PROGRAM P20_ExhaustFan_old
VAR
		(*****************Wentylator wyciągaowy*******************)
	fbExhaustFan							: FB_MitsubishiInverter;
	fbSensorAcetone							: FB_SensorAcetone;
	fbSensorAirFlow							: FB_SensorFlow;
	
	eExhaustFanState						: E_Station;			
	eExhaustFanRunningState					: E_ConveyorState;	
	fbExhaustFanState						: FB_State;		
	QnExhaustFanVelocitySV					AT %Q*: UDINT; 			(*po kom*)	// Nastawa prędkości transportera
	InExhaustFanVelocityCV 					AT %I*: UDINT;			(*po kom*)
	InExhaustFanSTW 						AT %I*: UINT; 			(*po kom*)	// Statusword transportera wejściowego
	QnExhaustFanCTW 						AT %Q*: UINT;  			(*po kom*)	// Controlword transportera wejsciowego
	InExhaustFanErrorCode 					AT %I*: UINT;			(*po kom*)

	(*** Detekcja acetonu***)
	IbSensorAcetoneDetectionNotError			AT %I* :BOOL;			//Czujnik detekcji acetonu usterka bład
	IbSensorAcetoneDetectionNotLevel2			AT %I* :BOOL;			// Alarm poziomu 2 detekcja acetonu 40%DGW (dolna granica wybuchowści)
	IbSensorAcetoneDetectionNotLevel1			AT %I* :BOOL;			// Alarm poziomu 1 detekcja acetonu 20%DGW (dolna granica wybuchowści)

	QbSensorAcetoneDetectionErrorSafety		AT %Q* :BOOL;			//Czujnik detekcji acetonu usterka bład
	QbSensorAcetoneDetectionLevel2Safety	AT %Q* :BOOL;			// Alarm poziomu 2 detekcja acetonu 40%DGW (dolna granica wybuchowści)
	//IbSensorAcetoneDetectionLevel1Safety	AT %Q* :BOOL;			// Alarm poziomu 1 detekcja acetonu 10%DGW (dolna granica wybuchowści)
	
	(*** Detekcja przepływu powietrza***)
	IbSensorFlowDetectionOK					AT %I* :BOOL;			// Czujnik przepływu powietrza - obencości przepłwu
	IbSensorFlowDetectionError				AT %I* :BOOL;			// Czujnik przepływu powietrza - błąd, alarm
	
	tofbExhaustFanCmdStartDelay: TOF;
	bExTest:BOOL;
END_VAR

aFan();
aSensors();

IF GVL_IO.IbExModeSwitchExMode THEN // SAFETY - PRZEPISANIE
	QbSensorAcetoneDetectionLevel2Safety	:=	IbSensorAcetoneDetectionNotLevel2;
	QbSensorAcetoneDetectionErrorSafety		:=	IbSensorAcetoneDetectionNotError;
ELSE 
	QbSensorAcetoneDetectionLevel2Safety	:=	TRUE;//FALSE;
	QbSensorAcetoneDetectionErrorSafety		:=	TRUE;
END_IF;

IF NOT IbSensorAcetoneDetectionNotLevel1 THEN
	udiExhaustFanVelocitySV:=1500;
ELSE
	udiExhaustFanVelocitySV:=750;
END_IF

VIS.udiExhaustFanVelocityCV:=InExhaustFanVelocityCV; //WIZKA

tofbExhaustFanCmdStartDelay(IN:= bExEnable AND NOT GVL.SensorAcetoneError.bError, PT:=T#3M);
tofbExhaustFanCmdStartDelay.ET;

IF NOT tofbExhaustFanCmdStartDelay.Q THEN
	bExhaustFanEnable		:= FALSE;	
	bExhaustFanCmdStart		:= FALSE;
END_IF

IF bExEnable THEN
	bExhaustFanEnable		:= TRUE;
	bExhaustFanCmdStart		:= TRUE;
END_IF

(*fbExhaustFanState(
	eState													:= eExhaustFanState , 
	bRun													:= bExhaustFanCmdStart,	
	eConveyorRunningState									:= eExhaustFanRunningState , 
	sStateDesc												=> VIS.sExhausFanState,
	iState													=> VIS.iExhausFanState	);*)
	
// Obsługa ostrzeżenia
ExSensorWarning[1].sDescription:=fbSensorAcetone.sWarningDescription;

IF (fbSensorAcetone.bWarning ) AND NOT ExSensorWarning[1].bWarning THEN
	ExSensorWarning[1].bWarning		:=	TRUE;
ELSIF ( NOT fbSensorAcetone.bWarning )AND ExSensorWarning[1].bAcknowledge THEN
	ExSensorWarning[1].bWarning		:=	FALSE;
	ExSensorWarning[1].bAcknowledge	:=	FALSE;
	VIS.uliWarningAcknowledge.24 	:=	FALSE;
ELSIF ExSensorWarning[1].bAcknowledge THEN
	ExSensorWarning[1].bAcknowledge	:=	TRUE;
END_IF

ACTION aFan:
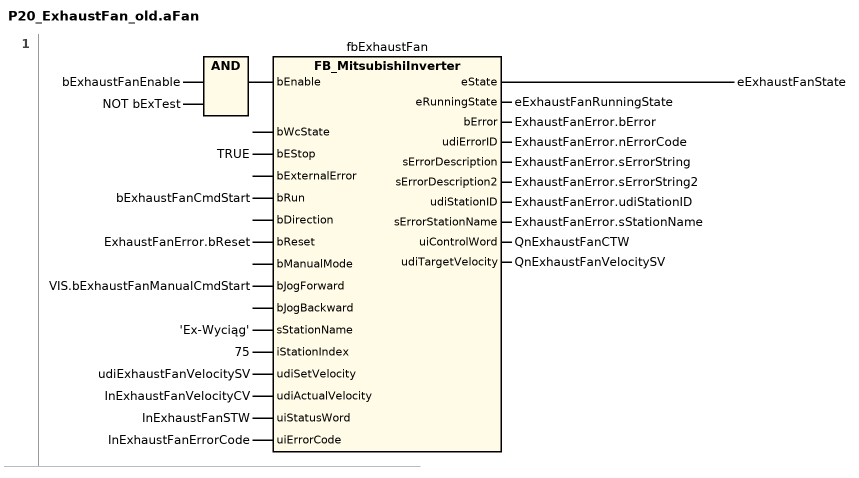
// NETWORK 1
fbExhaustFan(
    bEnable := bExhaustFanEnable AND (NOT bExTest),
    bEStop := TRUE,
    bRun := bExhaustFanCmdStart,
    bReset := ExhaustFanError.bReset,
    bJogForward := VIS.bExhaustFanManualCmdStart,
    sStationName := 'Ex-Wyciąg',
    iStationIndex := 75,
    udiSetVelocity := udiExhaustFanVelocitySV,
    udiActualVelocity := InExhaustFanVelocityCV,
    uiStatusWord := InExhaustFanSTW,
    uiErrorCode := InExhaustFanErrorCode,
    eRunningState => eExhaustFanRunningState,
    bError => ExhaustFanError.bError,
    udiErrorID => ExhaustFanError.nErrorCode,
    sErrorDescription => ExhaustFanError.sErrorString,
    sErrorDescription2 => ExhaustFanError.sErrorString2,
    udiStationID => ExhaustFanError.udiStationID,
    sErrorStationName => ExhaustFanError.sStationName,
    uiControlWord => QnExhaustFanCTW,
    udiTargetVelocity => QnExhaustFanVelocitySV); // FB_MitsubishiInverter
eExhaustFanState := fbExhaustFan.eState;
END_ACTION

ACTION aSensors:
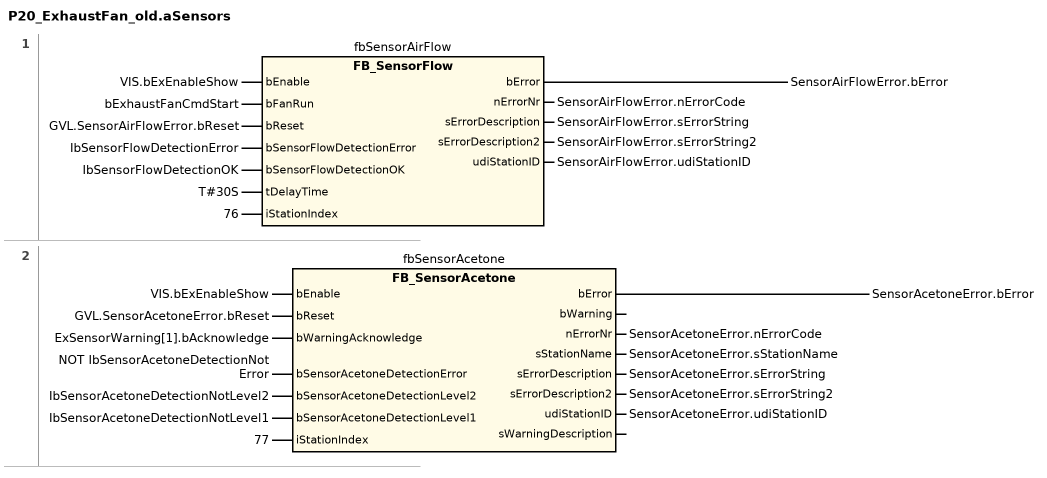
// NETWORK 1
fbSensorAirFlow(
    bEnable := VIS.bExEnableShow,
    bFanRun := bExhaustFanCmdStart,
    bReset := GVL.SensorAirFlowError.bReset,
    bSensorFlowDetectionError := IbSensorFlowDetectionError,
    bSensorFlowDetectionOK := IbSensorFlowDetectionOK,
    tDelayTime := T#30S,
    iStationIndex := 76,
    nErrorNr => SensorAirFlowError.nErrorCode,
    sErrorDescription => SensorAirFlowError.sErrorString,
    sErrorDescription2 => SensorAirFlowError.sErrorString2,
    udiStationID => SensorAirFlowError.udiStationID); // FB_SensorFlow
SensorAirFlowError.bError := fbSensorAirFlow.bError;

// NETWORK 2
fbSensorAcetone(
    bEnable := VIS.bExEnableShow,
    bReset := GVL.SensorAcetoneError.bReset,
    bWarningAcknowledge := ExSensorWarning[1].bAcknowledge,
    bSensorAcetoneDetectionError := NOT IbSensorAcetoneDetectionNotError,
    bSensorAcetoneDetectionLevel2 := IbSensorAcetoneDetectionNotLevel2,
    bSensorAcetoneDetectionLevel1 := IbSensorAcetoneDetectionNotLevel1,
    iStationIndex := 77,
    nErrorNr => SensorAcetoneError.nErrorCode,
    sStationName => SensorAcetoneError.sStationName,
    sErrorDescription => SensorAcetoneError.sErrorString,
    sErrorDescription2 => SensorAcetoneError.sErrorString2,
    udiStationID => SensorAcetoneError.udiStationID); // FB_SensorAcetone
SensorAcetoneError.bError := fbSensorAcetone.bError;
END_ACTION

END_PROGRAM

(* stored: Version 1.1.0.1, ProductVersion 3.1.4026.13, FileIdentifier 3fe324d9f701d50392390b8b92041315559d3290, FileSignature 370f0c974688adedb99b3f0d56236de3be753b300b2be6526accdb0772aa5daac87270c4408a468de09454e60df5c2a3dbb29839e7ce10b894de9ccefcbe8727ffb66927f8fe9efd779a84ec4efd6b3f6f8e636baf4003c6f1049cb0e1fd8f3f7588d4f4010284b61300704adc58781d6144a6acac5855023cd65769cd17396d1ad03404c428d473329d4e5cd0ab59302b3e106b2c8fbb5ab088c59b831685b76e69f3b5dc2925216e6ab8af1b75b1d993e5ece0e41124d47eabbb953df86d4fc77aaf6011603905dcff7d014833fc81148d5cb17898401cc13a3ccc430566bd50c0a35c81bf19bbef17abcc360d88068ba66da372be2bf7407c8ce5280a4f78
   POU P20_ExhaustFan_old: Id {acfc6a99-347b-480a-be24-ea6b84fe974d}, SpecialFunc None
   Action aFan: Id {6c4a670d-4016-4757-b8cc-532bd37165ce}
   Action aSensors: Id {35039138-8c29-4c40-a45c-7c24cc4bfe2b} *)
